SUBAPPLICATION Softkey_IX_TO_logiBUS_QX (* Konvertierung Softkey IXA zu logiBUS QXA *)
  (* Standard: 61499-2; Description: Copyright (c) 2023 Meisterschulen am Ostbahnhof This program and the accompanying materials are made available under the terms of the Eclipse Public License 2.0 which is available at https://www.eclipse.org/legal/epl-2.0/ SPDX-License-Identifier: EPL-2.0 *)
  (* Version 1.0, 2026-01-15, Franz Höpfinger, Meisterschulen am Ostbahnhof, initial API and implementation and/or initial documentation *)
  PACKAGE MyLib::sys;
  IMPORT isobus::UT::Q::const::IDs::ID_NULL;
  IMPORT logiBUS::io::DQ::logiBUS_DO;
  IMPORT logiBUS::io::DQ::logiBUS_DO_S;
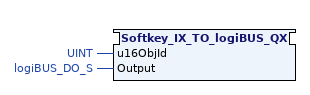
  VAR_INPUT
    u16ObjId : UINT := ID_NULL; (* Object ID *)
    Output : logiBUS::io::DQ::logiBUS_DO_S := logiBUS_DO::Invalid; (* Identify the Output Output_Q1..Q8 *)
  END_VAR
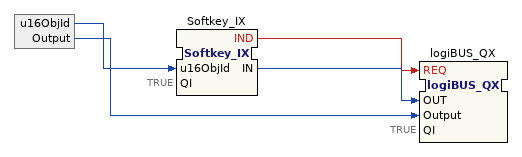
  FBS
    logiBUS_QX : logiBUS::io::DQ::logiBUS_QX(QI := TRUE);
    Softkey_IX : isobus::UT::io::Softkey::Softkey_IX(QI := TRUE);
  END_FBS
  EVENT_CONNECTIONS
    Softkey_IX.IND TO logiBUS_QX.REQ;
  END_CONNECTIONS
  DATA_CONNECTIONS
    Softkey_IX.IN TO logiBUS_QX.OUT;
    u16ObjId TO Softkey_IX.u16ObjId;
    Output TO logiBUS_QX.Output;
  END_CONNECTIONS
END_SUBAPPLICATION
